SPLINE
SPL {X  -149.193, Y  +319.722, Z    +0.000, E1   +76.912, E3 +131571.129}
SPL {X  -149.265, Y  +319.910, Z    +0.000, E1   +76.148, E3 +131579.729}
ENDSPLINE

SPLINE
SPL {X  -149.092, Y  +319.462, Z    +0.000, E1   +75.437, E3 +131587.604}
ENDSPLINE

SPLINE
SPL {X  -149.679, Y  +320.993, Z    +0.000, E1   +74.493, E3 +131596.498}
SPL {X  -149.823, Y  +321.377, Z    +0.000, E1   +73.518, E3 +131605.855}
ENDSPLINE

SPLINE
SPL {X  -149.061, Y  +319.382, Z    +0.000, E1   +72.547, E3 +131616.097}
SPL {X  -148.201, Y  +317.223, Z    +0.000, E1   +71.184, E3 +131629.421}
SPL {X  -144.085, Y  +307.957, Z    +0.000, E1   +70.311, E3 +131642.668}
SPL {X  -139.769, Y  +299.645, Z    +0.000, E1   +69.722, E3 +131652.399}
SPL {X  -136.083, Y  +293.369, Z    +0.000, E1   +69.227, E3 +131659.940}
SPL {X  -132.274, Y  +287.498, Z    +0.000, E1   +68.678, E3 +131667.159}
SPL {X  -128.237, Y  +281.834, Z    +0.000, E1   +68.080, E3 +131674.196}
SPL {X  -124.030, Y  +276.439, Z    +0.000, E1   +67.412, E3 +131680.913}
SPL {X   -89.505, Y  +244.889, Z    +0.000, E1   +58.168, E3 +131762.665}
ENDSPLINE

SPLINE
SPL {X  -111.763, Y  +263.019, Z    +0.000, E1   +52.505, E3 +131944.077}
SPL {X  -139.943, Y  +299.958, Z    +0.000, E1   +46.517, E3 +131978.417}
SPL {X  -154.122, Y  +334.569, Z    +0.000, E1   +33.405, E3 +131990.252}
SPL {X  -159.233, Y  +361.951, Z    +0.000, E1   +15.631, E3 +131994.430}
SPL {X  -159.983, Y  +375.952, Z    +0.000, E1    +3.555, E3 +131995.197}
SPL {X  -159.990, Y  +379.545, Z    +0.000, E1    -0.045, E3 +131995.243}
SPL {X  -159.990, Y  +382.058, Z    +0.000, E1    -4.728, E3 +131995.275}
SPL {X  -159.990, Y  +387.492, Z    +0.000, E1   -16.478, E3 +131995.501}
SPL {X  -159.990, Y  +395.172, Z    +0.000, E1   -33.361, E3 +131996.127}
SPL {X  -159.990, Y  +403.640, Z    +0.000, E1   -46.960, E3 +131997.275}
SPL {X  -159.990, Y  +418.500, Z    +0.000, E1   -59.260, E3 +132000.631}
SPL {X  -159.990, Y  +491.183, Z    +0.000, E1   -70.406, E3 +132028.312}
SPL {X  -159.990, Y  +644.105, Z    +0.000, E1   -71.828, E3 +132112.880}
SPL {X  -159.990, Y  +665.410, Z    +0.000, E1   -71.813, E3 +132127.778}
SPL {X  -159.784, Y  +684.619, Z    +0.000, E1   -71.795, E3 +132141.381}
SPL {X  -158.321, Y  +699.551, Z    +0.000, E1   -71.633, E3 +132153.333}
SPL {X  -155.878, Y  +712.540, Z    +0.000, E1   -71.376, E3 +132164.897}
SPL {X  -152.746, Y  +724.097, Z    +0.000, E1   -71.019, E3 +132176.148}
SPL {X  -149.840, Y  +732.578, Z    +0.000, E1   -70.669, E3 +132184.973}
SPL {X  -147.044, Y  +739.548, Z    +0.000, E1   -70.332, E3 +132192.567}
SPL {X  -143.437, Y  +747.371, Z    +0.000, E1   -69.890, E3 +132201.431}
SPL {X  -139.209, Y  +755.353, Z    +0.000, E1   -69.333, E3 +132210.858}
SPL {X  -135.354, Y  +761.800, Z    +0.000, E1   -68.789, E3 +132218.722}
SPL {X  -131.547, Y  +767.562, Z    +0.000, E1   -68.238, E3 +132225.891}
SPL {X  -127.113, Y  +773.655, Z    +0.000, E1   -67.565, E3 +132233.547}
SPL {X  -123.626, Y  +778.056, Z    +0.000, E1   -66.969, E3 +132239.107}
SPL {X   -86.110, Y  +811.340, Z    +0.000, E1   -55.142, E3 +132357.018}
ENDSPLINE

SPLINE
SPL {X  -126.688, Y  +774.208, Z    +0.000, E1   -50.278, E3 +132517.665}
SPL {X  -147.153, Y  +739.291, Z    +0.000, E1   -41.559, E3 +132538.500}
SPL {X  -156.578, Y  +709.366, Z    +0.000, E1   -27.394, E3 +132546.192}
SPL {X  -159.560, Y  +688.227, Z    +0.000, E1   -12.334, E3 +132548.757}
SPL {X  -159.987, Y  +677.470, Z    +0.000, E1    -2.943, E3 +132549.236}
SPL {X  -159.990, Y  +674.465, Z    +0.000, E1    +0.035, E3 +132549.268}
SPL {X  -159.990, Y  +672.210, Z    +0.000, E1    +4.112, E3 +132549.295}
SPL {X  -159.990, Y  +668.446, Z    +0.000, E1   +12.084, E3 +132549.420}
SPL {X  -159.990, Y  +663.424, Z    +0.000, E1   +23.273, E3 +132549.747}
SPL {X  -159.990, Y  +655.288, Z    +0.000, E1   +39.016, E3 +132550.636}
SPL {X  -159.990, Y  +641.020, Z    +0.000, E1   +55.512, E3 +132553.175}
SPL {X  -159.990, Y  +618.237, Z    +0.000, E1   +65.205, E3 +132559.700}
SPL {X  -159.990, Y  +545.807, Z    +0.000, E1   +71.095, E3 +132588.753}
SPL {X  -159.990, Y  +417.971, Z    +0.000, E1   +72.138, E3 +132657.413}
SPL {X  -147.674, Y  +315.943, Z    +0.000, E1   +77.803, E3 +132649.143}
ENDSPLINE

SPLINE
SPL {X  -149.193, Y  +319.722, Z    +0.000, E1   +76.912, E3 +132658.085}
ENDSPLINE

SPLINE
SPL {X  -149.153, Y  +319.620, Z    +0.000, E1   +75.840, E3 +132670.495}
ENDSPLINE

SPLINE
SPL {X  -149.679, Y  +320.993, Z    +0.000, E1   +74.493, E3 +132683.454}
SPL {X  -149.823, Y  +321.377, Z    +0.000, E1   +73.518, E3 +132692.812}
ENDSPLINE

SPLINE
SPL {X  -149.061, Y  +319.382, Z    +0.000, E1   +72.547, E3 +132703.053}
SPL {X  -148.522, Y  +318.020, Z    +0.000, E1   +71.446, E3 +132713.439}
ENDSPLINE

SLIN {X  -200.000, Y  +530.000, E1    +0.000}
HALT
END
